PROGRAM MAIN
VAR
END_VAR

END_PROGRAM

(* stored: Version 1.1.0.1
   POU MAIN: Id {2e728b70-dd3c-4ef0-af6f-a5f63b404be7} *)
